REGION Network 174: Reset CV hơi Bồn 4 khi không chạy PID
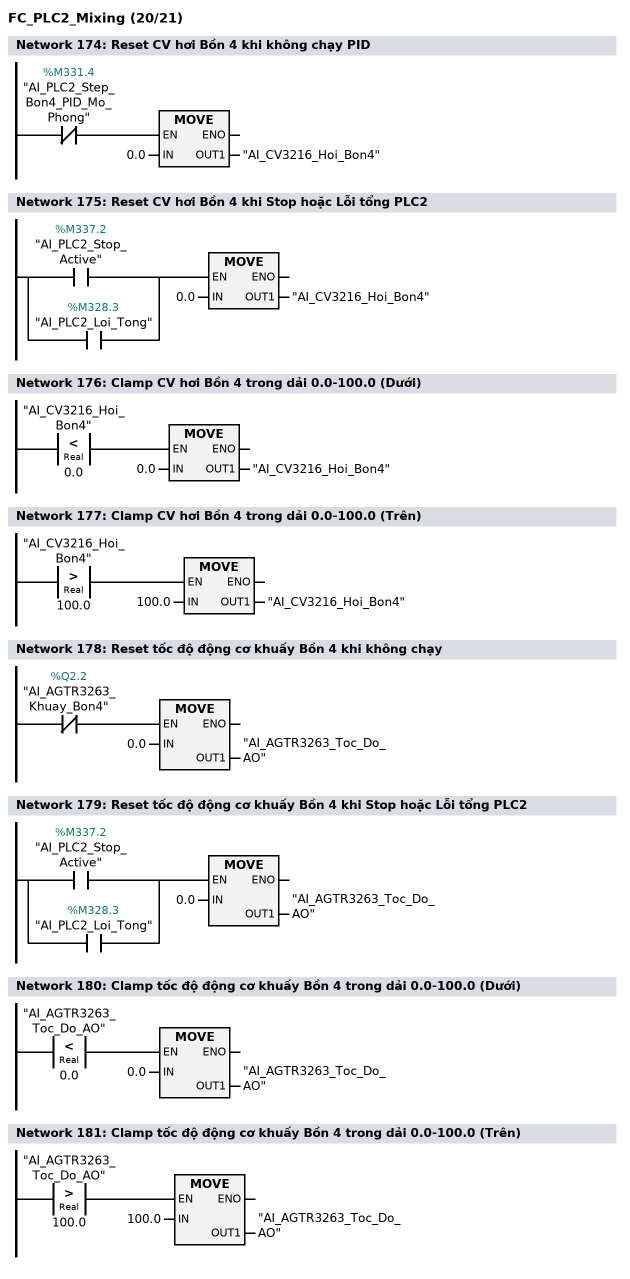
   RUNG wire#powerrail
      I_Contact( "AI_PLC2_Step_Bon4_PID_Mo_Phong" )
      { S7_GenerateENO := "TRUE" } Move(in := 0.0, out1 => "AI_CV3216_Hoi_Bon4")
   END_RUNG
   // the same network as SCL:
   IF NOT "AI_PLC2_Step_Bon4_PID_Mo_Phong" THEN "AI_CV3216_Hoi_Bon4" := 0.0; END_IF;
END_REGION

REGION Network 175: Reset CV hơi Bồn 4 khi Stop hoặc Lỗi tổng PLC2
   RUNG wire#powerrail
      Contact( "AI_PLC2_Stop_Active" )
      wire#w1
      { S7_GenerateENO := "TRUE" } Move(in := 0.0, out1 => "AI_CV3216_Hoi_Bon4")
   END_RUNG
   RUNG wire#powerrail
      Contact( "AI_PLC2_Loi_Tong" )
   END_RUNG wire#w1
   // the same network as SCL:
   IF "AI_PLC2_Stop_Active" OR "AI_PLC2_Loi_Tong" THEN "AI_CV3216_Hoi_Bon4" := 0.0; END_IF;
END_REGION

REGION Network 176: Clamp CV hơi Bồn 4 trong dải 0.0-100.0 (Dưới)
   RUNG wire#powerrail
      { S7_Templates := "SrcType := Real" } LT_Contact(in1 := "AI_CV3216_Hoi_Bon4", in2 := 0.0)
      { S7_GenerateENO := "TRUE" } Move(in := 0.0, out1 => "AI_CV3216_Hoi_Bon4")
   END_RUNG
   // the same network as SCL:
   IF "AI_CV3216_Hoi_Bon4" < 0.0 THEN "AI_CV3216_Hoi_Bon4" := 0.0; END_IF;
END_REGION

REGION Network 177: Clamp CV hơi Bồn 4 trong dải 0.0-100.0 (Trên)
   RUNG wire#powerrail
      { S7_Templates := "SrcType := Real" } GT_Contact(in1 := "AI_CV3216_Hoi_Bon4", in2 := 100.0)
      { S7_GenerateENO := "TRUE" } Move(in := 100.0, out1 => "AI_CV3216_Hoi_Bon4")
   END_RUNG
   // the same network as SCL:
   IF "AI_CV3216_Hoi_Bon4" > 100.0 THEN "AI_CV3216_Hoi_Bon4" := 100.0; END_IF;
END_REGION

REGION Network 178: Reset tốc độ động cơ khuấy Bồn 4 khi không chạy
   RUNG wire#powerrail
      I_Contact( "AI_AGTR3263_Khuay_Bon4" )
      { S7_GenerateENO := "TRUE" } Move(in := 0.0, out1 => "AI_AGTR3263_Toc_Do_AO")
   END_RUNG
   // the same network as SCL:
   IF NOT "AI_AGTR3263_Khuay_Bon4" THEN "AI_AGTR3263_Toc_Do_AO" := 0.0; END_IF;
END_REGION

REGION Network 179: Reset tốc độ động cơ khuấy Bồn 4 khi Stop hoặc Lỗi tổng PLC2
   RUNG wire#powerrail
      Contact( "AI_PLC2_Stop_Active" )
      wire#w1
      { S7_GenerateENO := "TRUE" } Move(in := 0.0, out1 => "AI_AGTR3263_Toc_Do_AO")
   END_RUNG
   RUNG wire#powerrail
      Contact( "AI_PLC2_Loi_Tong" )
   END_RUNG wire#w1
   // the same network as SCL:
   IF "AI_PLC2_Stop_Active" OR "AI_PLC2_Loi_Tong" THEN "AI_AGTR3263_Toc_Do_AO" := 0.0; END_IF;
END_REGION

REGION Network 180: Clamp tốc độ động cơ khuấy Bồn 4 trong dải 0.0-100.0 (Dưới)
   RUNG wire#powerrail
      { S7_Templates := "SrcType := Real" } LT_Contact(in1 := "AI_AGTR3263_Toc_Do_AO", in2 := 0.0)
      { S7_GenerateENO := "TRUE" } Move(in := 0.0, out1 => "AI_AGTR3263_Toc_Do_AO")
   END_RUNG
   // the same network as SCL:
   IF "AI_AGTR3263_Toc_Do_AO" < 0.0 THEN "AI_AGTR3263_Toc_Do_AO" := 0.0; END_IF;
END_REGION

REGION Network 181: Clamp tốc độ động cơ khuấy Bồn 4 trong dải 0.0-100.0 (Trên)
   RUNG wire#powerrail
      { S7_Templates := "SrcType := Real" } GT_Contact(in1 := "AI_AGTR3263_Toc_Do_AO", in2 := 100.0)
      { S7_GenerateENO := "TRUE" } Move(in := 100.0, out1 => "AI_AGTR3263_Toc_Do_AO")
   END_RUNG
   // the same network as SCL:
   IF "AI_AGTR3263_Toc_Do_AO" > 100.0 THEN "AI_AGTR3263_Toc_Do_AO" := 100.0; END_IF;
END_REGION

REGION Network 182: Dừng an toàn PLC2 reset AI_V3240_Nuoc_Bon3
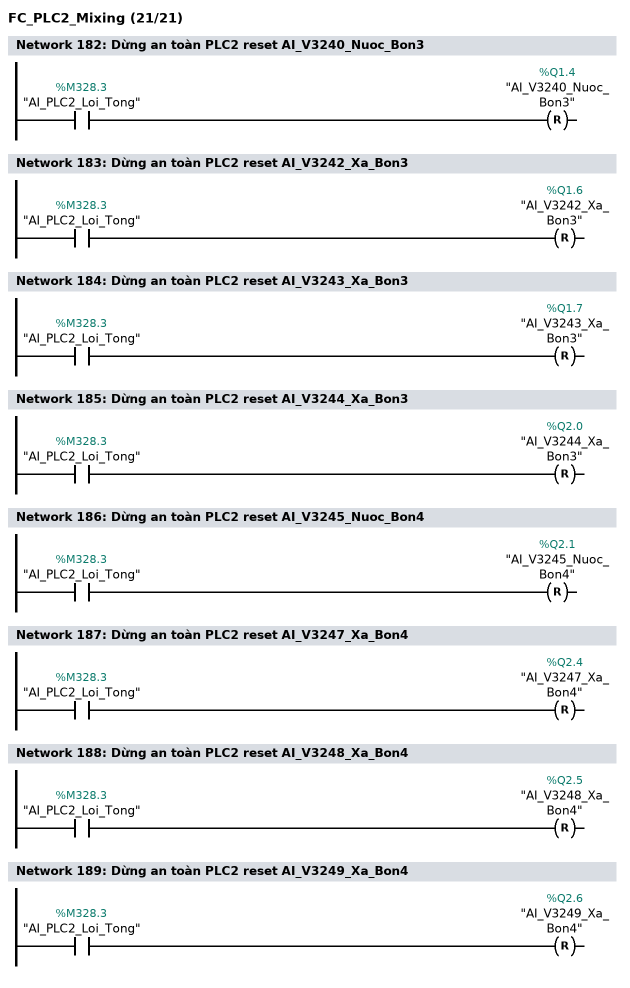
   RUNG wire#powerrail
      Contact( "AI_PLC2_Loi_Tong" )
      R_Coil( "AI_V3240_Nuoc_Bon3" )
   END_RUNG
   // the same network as SCL:
   IF "AI_PLC2_Loi_Tong" THEN "AI_V3240_Nuoc_Bon3" := FALSE; END_IF;
END_REGION

REGION Network 183: Dừng an toàn PLC2 reset AI_V3242_Xa_Bon3
   RUNG wire#powerrail
      Contact( "AI_PLC2_Loi_Tong" )
      R_Coil( "AI_V3242_Xa_Bon3" )
   END_RUNG
   // the same network as SCL:
   IF "AI_PLC2_Loi_Tong" THEN "AI_V3242_Xa_Bon3" := FALSE; END_IF;
END_REGION

REGION Network 184: Dừng an toàn PLC2 reset AI_V3243_Xa_Bon3
   RUNG wire#powerrail
      Contact( "AI_PLC2_Loi_Tong" )
      R_Coil( "AI_V3243_Xa_Bon3" )
   END_RUNG
   // the same network as SCL:
   IF "AI_PLC2_Loi_Tong" THEN "AI_V3243_Xa_Bon3" := FALSE; END_IF;
END_REGION

REGION Network 185: Dừng an toàn PLC2 reset AI_V3244_Xa_Bon3
   RUNG wire#powerrail
      Contact( "AI_PLC2_Loi_Tong" )
      R_Coil( "AI_V3244_Xa_Bon3" )
   END_RUNG
   // the same network as SCL:
   IF "AI_PLC2_Loi_Tong" THEN "AI_V3244_Xa_Bon3" := FALSE; END_IF;
END_REGION

REGION Network 186: Dừng an toàn PLC2 reset AI_V3245_Nuoc_Bon4
   RUNG wire#powerrail
      Contact( "AI_PLC2_Loi_Tong" )
      R_Coil( "AI_V3245_Nuoc_Bon4" )
   END_RUNG
   // the same network as SCL:
   IF "AI_PLC2_Loi_Tong" THEN "AI_V3245_Nuoc_Bon4" := FALSE; END_IF;
END_REGION

REGION Network 187: Dừng an toàn PLC2 reset AI_V3247_Xa_Bon4
   RUNG wire#powerrail
      Contact( "AI_PLC2_Loi_Tong" )
      R_Coil( "AI_V3247_Xa_Bon4" )
   END_RUNG
   // the same network as SCL:
   IF "AI_PLC2_Loi_Tong" THEN "AI_V3247_Xa_Bon4" := FALSE; END_IF;
END_REGION

REGION Network 188: Dừng an toàn PLC2 reset AI_V3248_Xa_Bon4
   RUNG wire#powerrail
      Contact( "AI_PLC2_Loi_Tong" )
      R_Coil( "AI_V3248_Xa_Bon4" )
   END_RUNG
   // the same network as SCL:
   IF "AI_PLC2_Loi_Tong" THEN "AI_V3248_Xa_Bon4" := FALSE; END_IF;
END_REGION

REGION Network 189: Dừng an toàn PLC2 reset AI_V3249_Xa_Bon4
   RUNG wire#powerrail
      Contact( "AI_PLC2_Loi_Tong" )
      R_Coil( "AI_V3249_Xa_Bon4" )
   END_RUNG
   // the same network as SCL:
   IF "AI_PLC2_Loi_Tong" THEN "AI_V3249_Xa_Bon4" := FALSE; END_IF;
END_REGION
END_FUNCTION

FUNCTION "FC_HMI_Mirror_PLC2" : Void   // FC41, LAD
{ S7_Optimized_Access := 'TRUE' }
VERSION : 0.1
// stored: AutoNumber true, IsIECCheckEnabled false, SetENOAutomatically false, UDAEnableTagReadback false
BEGIN

REGION Network 1: Mirror AI_V3240_Nuoc_Bon3
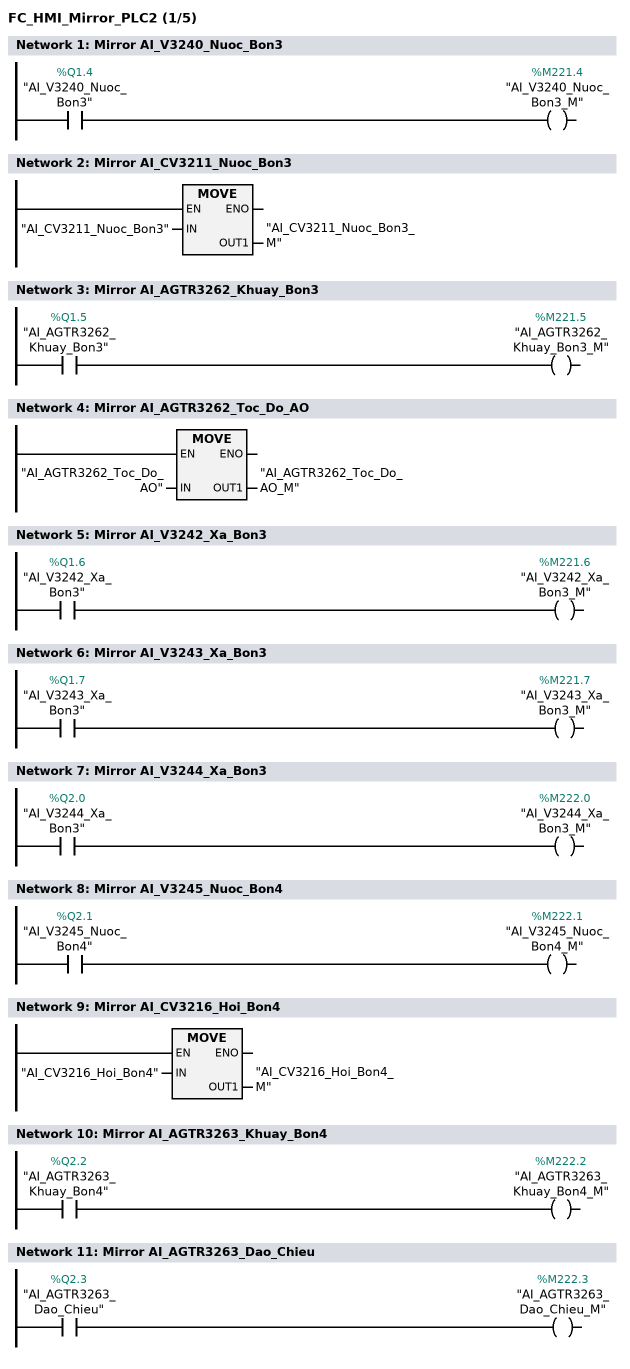
   RUNG wire#powerrail
      Contact( "AI_V3240_Nuoc_Bon3" )
      Coil( "AI_V3240_Nuoc_Bon3_M" )
   END_RUNG
   // the same network as SCL:
   "AI_V3240_Nuoc_Bon3_M" := "AI_V3240_Nuoc_Bon3";
END_REGION

REGION Network 2: Mirror AI_CV3211_Nuoc_Bon3
   RUNG wire#powerrail
      { S7_GenerateENO := "TRUE" } Move(in := "AI_CV3211_Nuoc_Bon3", out1 => "AI_CV3211_Nuoc_Bon3_M")
   END_RUNG
   // the same network as SCL:
   "AI_CV3211_Nuoc_Bon3_M" := "AI_CV3211_Nuoc_Bon3";
END_REGION

REGION Network 3: Mirror AI_AGTR3262_Khuay_Bon3
   RUNG wire#powerrail
      Contact( "AI_AGTR3262_Khuay_Bon3" )
      Coil( "AI_AGTR3262_Khuay_Bon3_M" )
   END_RUNG
   // the same network as SCL:
   "AI_AGTR3262_Khuay_Bon3_M" := "AI_AGTR3262_Khuay_Bon3";
END_REGION

REGION Network 4: Mirror AI_AGTR3262_Toc_Do_AO
   RUNG wire#powerrail
      { S7_GenerateENO := "TRUE" } Move(in := "AI_AGTR3262_Toc_Do_AO", out1 => "AI_AGTR3262_Toc_Do_AO_M")
   END_RUNG
   // the same network as SCL:
   "AI_AGTR3262_Toc_Do_AO_M" := "AI_AGTR3262_Toc_Do_AO";
END_REGION

REGION Network 5: Mirror AI_V3242_Xa_Bon3
   RUNG wire#powerrail
      Contact( "AI_V3242_Xa_Bon3" )
      Coil( "AI_V3242_Xa_Bon3_M" )
   END_RUNG
   // the same network as SCL:
   "AI_V3242_Xa_Bon3_M" := "AI_V3242_Xa_Bon3";
END_REGION

REGION Network 6: Mirror AI_V3243_Xa_Bon3
   RUNG wire#powerrail
      Contact( "AI_V3243_Xa_Bon3" )
      Coil( "AI_V3243_Xa_Bon3_M" )
   END_RUNG
   // the same network as SCL:
   "AI_V3243_Xa_Bon3_M" := "AI_V3243_Xa_Bon3";
END_REGION

REGION Network 7: Mirror AI_V3244_Xa_Bon3
   RUNG wire#powerrail
      Contact( "AI_V3244_Xa_Bon3" )
      Coil( "AI_V3244_Xa_Bon3_M" )
   END_RUNG
   // the same network as SCL:
   "AI_V3244_Xa_Bon3_M" := "AI_V3244_Xa_Bon3";
END_REGION

REGION Network 8: Mirror AI_V3245_Nuoc_Bon4
   RUNG wire#powerrail
      Contact( "AI_V3245_Nuoc_Bon4" )
      Coil( "AI_V3245_Nuoc_Bon4_M" )
   END_RUNG
   // the same network as SCL:
   "AI_V3245_Nuoc_Bon4_M" := "AI_V3245_Nuoc_Bon4";
END_REGION

REGION Network 9: Mirror AI_CV3216_Hoi_Bon4
   RUNG wire#powerrail
      { S7_GenerateENO := "TRUE" } Move(in := "AI_CV3216_Hoi_Bon4", out1 => "AI_CV3216_Hoi_Bon4_M")
   END_RUNG
   // the same network as SCL:
   "AI_CV3216_Hoi_Bon4_M" := "AI_CV3216_Hoi_Bon4";
END_REGION

REGION Network 10: Mirror AI_AGTR3263_Khuay_Bon4
   RUNG wire#powerrail
      Contact( "AI_AGTR3263_Khuay_Bon4" )
      Coil( "AI_AGTR3263_Khuay_Bon4_M" )
   END_RUNG
   // the same network as SCL:
   "AI_AGTR3263_Khuay_Bon4_M" := "AI_AGTR3263_Khuay_Bon4";
END_REGION

REGION Network 11: Mirror AI_AGTR3263_Dao_Chieu
   RUNG wire#powerrail
      Contact( "AI_AGTR3263_Dao_Chieu" )
      Coil( "AI_AGTR3263_Dao_Chieu_M" )
   END_RUNG
   // the same network as SCL:
   "AI_AGTR3263_Dao_Chieu_M" := "AI_AGTR3263_Dao_Chieu";
END_REGION

REGION Network 12: Mirror AI_AGTR3263_Toc_Do_AO
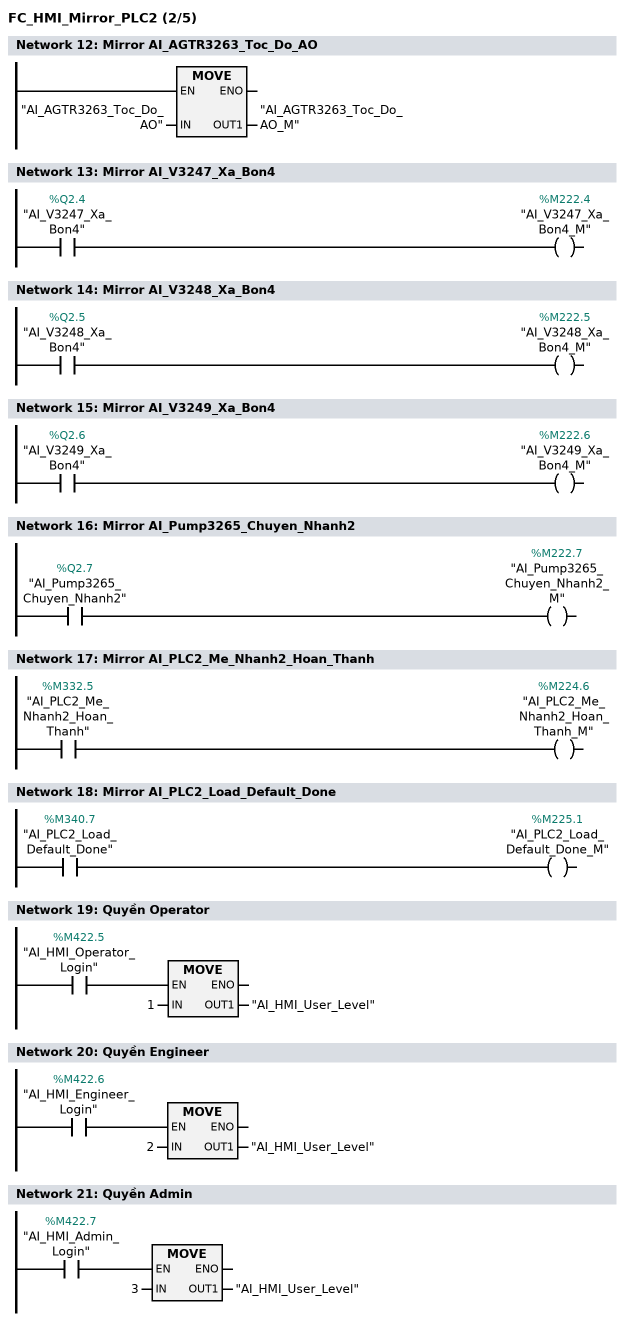
   RUNG wire#powerrail
      { S7_GenerateENO := "TRUE" } Move(in := "AI_AGTR3263_Toc_Do_AO", out1 => "AI_AGTR3263_Toc_Do_AO_M")
   END_RUNG
   // the same network as SCL:
   "AI_AGTR3263_Toc_Do_AO_M" := "AI_AGTR3263_Toc_Do_AO";
END_REGION

REGION Network 13: Mirror AI_V3247_Xa_Bon4
   RUNG wire#powerrail
      Contact( "AI_V3247_Xa_Bon4" )
      Coil( "AI_V3247_Xa_Bon4_M" )
   END_RUNG
   // the same network as SCL:
   "AI_V3247_Xa_Bon4_M" := "AI_V3247_Xa_Bon4";
END_REGION

REGION Network 14: Mirror AI_V3248_Xa_Bon4
   RUNG wire#powerrail
      Contact( "AI_V3248_Xa_Bon4" )
      Coil( "AI_V3248_Xa_Bon4_M" )
   END_RUNG
   // the same network as SCL:
   "AI_V3248_Xa_Bon4_M" := "AI_V3248_Xa_Bon4";
END_REGION

REGION Network 15: Mirror AI_V3249_Xa_Bon4
   RUNG wire#powerrail
      Contact( "AI_V3249_Xa_Bon4" )
      Coil( "AI_V3249_Xa_Bon4_M" )
   END_RUNG
   // the same network as SCL:
   "AI_V3249_Xa_Bon4_M" := "AI_V3249_Xa_Bon4";
END_REGION

REGION Network 16: Mirror AI_Pump3265_Chuyen_Nhanh2
   RUNG wire#powerrail
      Contact( "AI_Pump3265_Chuyen_Nhanh2" )
      Coil( "AI_Pump3265_Chuyen_Nhanh2_M" )
   END_RUNG
   // the same network as SCL:
   "AI_Pump3265_Chuyen_Nhanh2_M" := "AI_Pump3265_Chuyen_Nhanh2";
END_REGION

REGION Network 17: Mirror AI_PLC2_Me_Nhanh2_Hoan_Thanh
   RUNG wire#powerrail
      Contact( "AI_PLC2_Me_Nhanh2_Hoan_Thanh" )
      Coil( "AI_PLC2_Me_Nhanh2_Hoan_Thanh_M" )
   END_RUNG
   // the same network as SCL:
   "AI_PLC2_Me_Nhanh2_Hoan_Thanh_M" := "AI_PLC2_Me_Nhanh2_Hoan_Thanh";
END_REGION

REGION Network 18: Mirror AI_PLC2_Load_Default_Done
   RUNG wire#powerrail
      Contact( "AI_PLC2_Load_Default_Done" )
      Coil( "AI_PLC2_Load_Default_Done_M" )
   END_RUNG
   // the same network as SCL:
   "AI_PLC2_Load_Default_Done_M" := "AI_PLC2_Load_Default_Done";
END_REGION

REGION Network 19: Quyền Operator
   RUNG wire#powerrail
      Contact( "AI_HMI_Operator_Login" )
      { S7_GenerateENO := "TRUE" } Move(in := 1, out1 => "AI_HMI_User_Level")
   END_RUNG
   // the same network as SCL:
   IF "AI_HMI_Operator_Login" THEN "AI_HMI_User_Level" := 1; END_IF;
END_REGION

REGION Network 20: Quyền Engineer
   RUNG wire#powerrail
      Contact( "AI_HMI_Engineer_Login" )
      { S7_GenerateENO := "TRUE" } Move(in := 2, out1 => "AI_HMI_User_Level")
   END_RUNG
   // the same network as SCL:
   IF "AI_HMI_Engineer_Login" THEN "AI_HMI_User_Level" := 2; END_IF;
END_REGION

REGION Network 21: Quyền Admin
   RUNG wire#powerrail
      Contact( "AI_HMI_Admin_Login" )
      { S7_GenerateENO := "TRUE" } Move(in := 3, out1 => "AI_HMI_User_Level")
   END_RUNG
   // the same network as SCL:
   IF "AI_HMI_Admin_Login" THEN "AI_HMI_User_Level" := 3; END_IF;
END_REGION

REGION Network 22: Cho phép sửa thông số Engineer
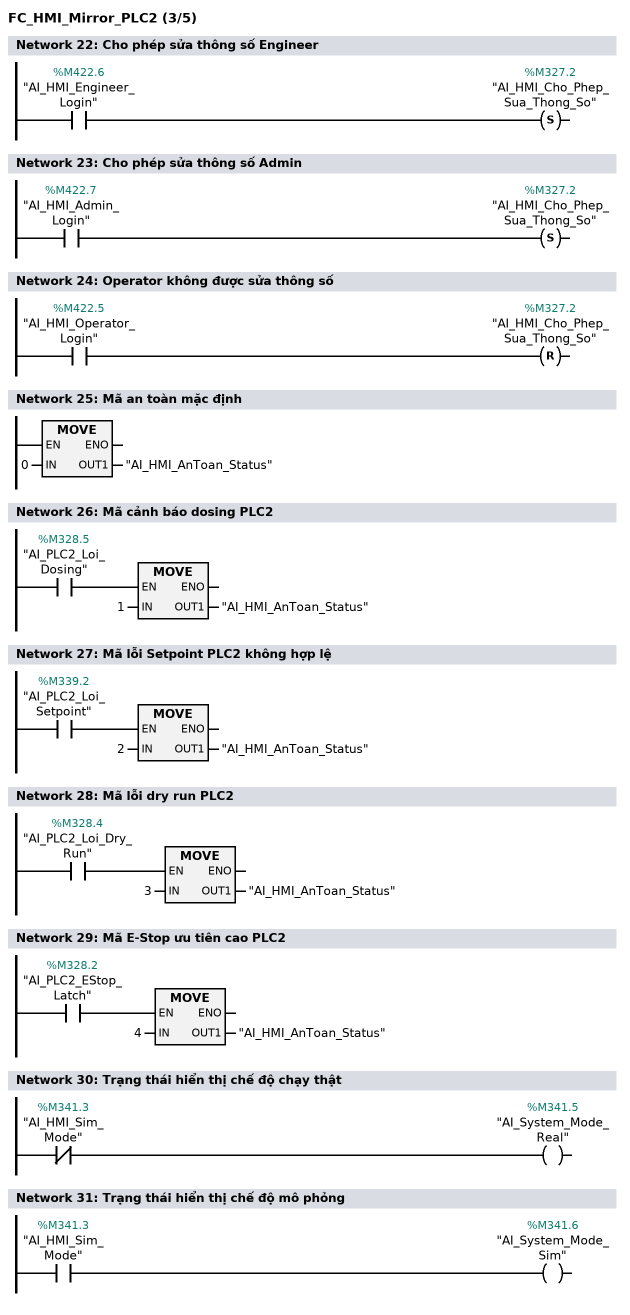
   RUNG wire#powerrail
      Contact( "AI_HMI_Engineer_Login" )
      S_Coil( "AI_HMI_Cho_Phep_Sua_Thong_So" )
   END_RUNG
   // the same network as SCL:
   IF "AI_HMI_Engineer_Login" THEN "AI_HMI_Cho_Phep_Sua_Thong_So" := TRUE; END_IF;
END_REGION

REGION Network 23: Cho phép sửa thông số Admin
   RUNG wire#powerrail
      Contact( "AI_HMI_Admin_Login" )
      S_Coil( "AI_HMI_Cho_Phep_Sua_Thong_So" )
   END_RUNG
   // the same network as SCL:
   IF "AI_HMI_Admin_Login" THEN "AI_HMI_Cho_Phep_Sua_Thong_So" := TRUE; END_IF;
END_REGION

REGION Network 24: Operator không được sửa thông số
   RUNG wire#powerrail
      Contact( "AI_HMI_Operator_Login" )
      R_Coil( "AI_HMI_Cho_Phep_Sua_Thong_So" )
   END_RUNG
   // the same network as SCL:
   IF "AI_HMI_Operator_Login" THEN "AI_HMI_Cho_Phep_Sua_Thong_So" := FALSE; END_IF;
END_REGION

REGION Network 25: Mã an toàn mặc định
   RUNG wire#powerrail
      { S7_GenerateENO := "TRUE" } Move(in := 0, out1 => "AI_HMI_AnToan_Status")
   END_RUNG
   // the same network as SCL:
   "AI_HMI_AnToan_Status" := 0;
END_REGION

REGION Network 26: Mã cảnh báo dosing PLC2
   RUNG wire#powerrail
      Contact( "AI_PLC2_Loi_Dosing" )
      { S7_GenerateENO := "TRUE" } Move(in := 1, out1 => "AI_HMI_AnToan_Status")
   END_RUNG
   // the same network as SCL:
   IF "AI_PLC2_Loi_Dosing" THEN "AI_HMI_AnToan_Status" := 1; END_IF;
END_REGION

REGION Network 27: Mã lỗi Setpoint PLC2 không hợp lệ
   RUNG wire#powerrail
      Contact( "AI_PLC2_Loi_Setpoint" )
      { S7_GenerateENO := "TRUE" } Move(in := 2, out1 => "AI_HMI_AnToan_Status")
   END_RUNG
   // the same network as SCL:
   IF "AI_PLC2_Loi_Setpoint" THEN "AI_HMI_AnToan_Status" := 2; END_IF;
END_REGION

REGION Network 28: Mã lỗi dry run PLC2
   RUNG wire#powerrail
      Contact( "AI_PLC2_Loi_Dry_Run" )
      { S7_GenerateENO := "TRUE" } Move(in := 3, out1 => "AI_HMI_AnToan_Status")
   END_RUNG
   // the same network as SCL:
   IF "AI_PLC2_Loi_Dry_Run" THEN "AI_HMI_AnToan_Status" := 3; END_IF;
END_REGION

REGION Network 29: Mã E-Stop ưu tiên cao PLC2
   RUNG wire#powerrail
      Contact( "AI_PLC2_EStop_Latch" )
      { S7_GenerateENO := "TRUE" } Move(in := 4, out1 => "AI_HMI_AnToan_Status")
   END_RUNG
   // the same network as SCL:
   IF "AI_PLC2_EStop_Latch" THEN "AI_HMI_AnToan_Status" := 4; END_IF;
END_REGION

REGION Network 30: Trạng thái hiển thị chế độ chạy thật
   RUNG wire#powerrail
      I_Contact( "AI_HMI_Sim_Mode" )
      Coil( "AI_System_Mode_Real" )
   END_RUNG
   // the same network as SCL:
   "AI_System_Mode_Real" := NOT "AI_HMI_Sim_Mode";
END_REGION

REGION Network 31: Trạng thái hiển thị chế độ mô phỏng
   RUNG wire#powerrail
      Contact( "AI_HMI_Sim_Mode" )
      Coil( "AI_System_Mode_Sim" )
   END_RUNG
   // the same network as SCL:
   "AI_System_Mode_Sim" := "AI_HMI_Sim_Mode";
END_REGION

REGION Network 32: Cảnh báo chế độ mô phỏng HMI active
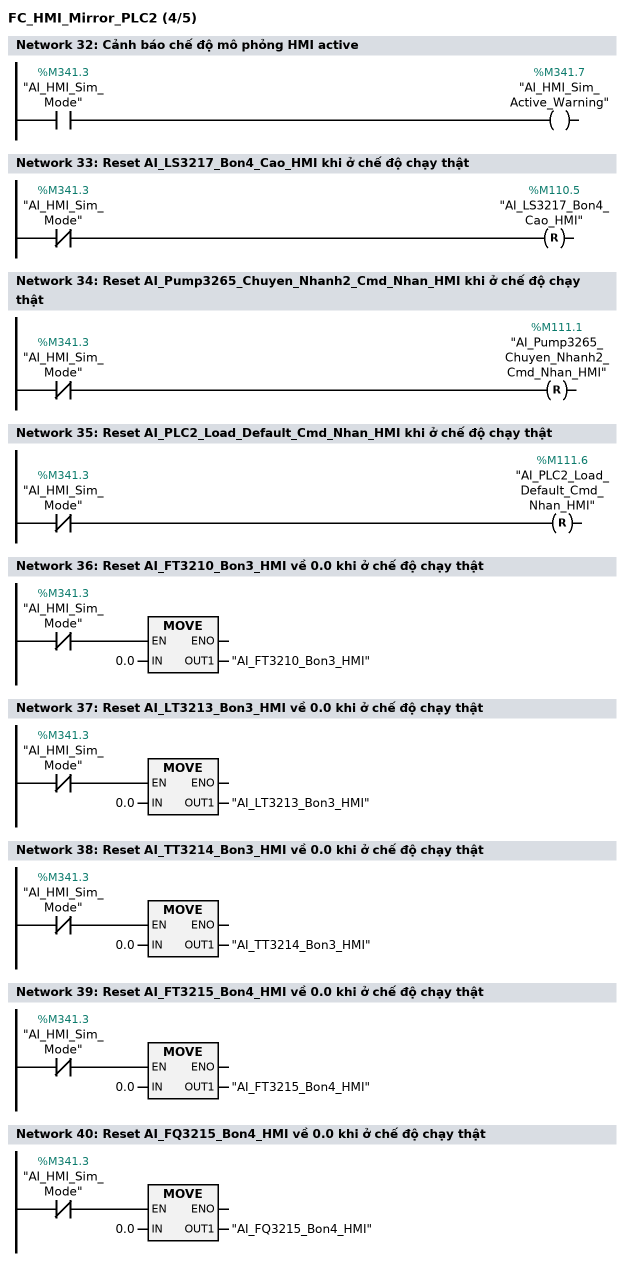
   RUNG wire#powerrail
      Contact( "AI_HMI_Sim_Mode" )
      Coil( "AI_HMI_Sim_Active_Warning" )
   END_RUNG
   // the same network as SCL:
   "AI_HMI_Sim_Active_Warning" := "AI_HMI_Sim_Mode";
END_REGION

REGION Network 33: Reset AI_LS3217_Bon4_Cao_HMI khi ở chế độ chạy thật
   RUNG wire#powerrail
      I_Contact( "AI_HMI_Sim_Mode" )
      R_Coil( "AI_LS3217_Bon4_Cao_HMI" )
   END_RUNG
   // the same network as SCL:
   IF NOT "AI_HMI_Sim_Mode" THEN "AI_LS3217_Bon4_Cao_HMI" := FALSE; END_IF;
END_REGION

REGION Network 34: Reset AI_Pump3265_Chuyen_Nhanh2_Cmd_Nhan_HMI khi ở chế độ chạy thật
   RUNG wire#powerrail
      I_Contact( "AI_HMI_Sim_Mode" )
      R_Coil( "AI_Pump3265_Chuyen_Nhanh2_Cmd_Nhan_HMI" )
   END_RUNG
   // the same network as SCL:
   IF NOT "AI_HMI_Sim_Mode" THEN "AI_Pump3265_Chuyen_Nhanh2_Cmd_Nhan_HMI" := FALSE; END_IF;
END_REGION

REGION Network 35: Reset AI_PLC2_Load_Default_Cmd_Nhan_HMI khi ở chế độ chạy thật
   RUNG wire#powerrail
      I_Contact( "AI_HMI_Sim_Mode" )
      R_Coil( "AI_PLC2_Load_Default_Cmd_Nhan_HMI" )
   END_RUNG
   // the same network as SCL:
   IF NOT "AI_HMI_Sim_Mode" THEN "AI_PLC2_Load_Default_Cmd_Nhan_HMI" := FALSE; END_IF;
END_REGION

REGION Network 36: Reset AI_FT3210_Bon3_HMI về 0.0 khi ở chế độ chạy thật
   RUNG wire#powerrail
      I_Contact( "AI_HMI_Sim_Mode" )
      { S7_GenerateENO := "TRUE" } Move(in := 0.0, out1 => "AI_FT3210_Bon3_HMI")
   END_RUNG
   // the same network as SCL:
   IF NOT "AI_HMI_Sim_Mode" THEN "AI_FT3210_Bon3_HMI" := 0.0; END_IF;
END_REGION

REGION Network 37: Reset AI_LT3213_Bon3_HMI về 0.0 khi ở chế độ chạy thật
   RUNG wire#powerrail
      I_Contact( "AI_HMI_Sim_Mode" )
      { S7_GenerateENO := "TRUE" } Move(in := 0.0, out1 => "AI_LT3213_Bon3_HMI")
   END_RUNG
   // the same network as SCL:
   IF NOT "AI_HMI_Sim_Mode" THEN "AI_LT3213_Bon3_HMI" := 0.0; END_IF;
END_REGION

REGION Network 38: Reset AI_TT3214_Bon3_HMI về 0.0 khi ở chế độ chạy thật
   RUNG wire#powerrail
      I_Contact( "AI_HMI_Sim_Mode" )
      { S7_GenerateENO := "TRUE" } Move(in := 0.0, out1 => "AI_TT3214_Bon3_HMI")
   END_RUNG
   // the same network as SCL:
   IF NOT "AI_HMI_Sim_Mode" THEN "AI_TT3214_Bon3_HMI" := 0.0; END_IF;
END_REGION

REGION Network 39: Reset AI_FT3215_Bon4_HMI về 0.0 khi ở chế độ chạy thật
   RUNG wire#powerrail
      I_Contact( "AI_HMI_Sim_Mode" )
      { S7_GenerateENO := "TRUE" } Move(in := 0.0, out1 => "AI_FT3215_Bon4_HMI")
   END_RUNG
   // the same network as SCL:
   IF NOT "AI_HMI_Sim_Mode" THEN "AI_FT3215_Bon4_HMI" := 0.0; END_IF;
END_REGION

REGION Network 40: Reset AI_FQ3215_Bon4_HMI về 0.0 khi ở chế độ chạy thật
   RUNG wire#powerrail
      I_Contact( "AI_HMI_Sim_Mode" )
      { S7_GenerateENO := "TRUE" } Move(in := 0.0, out1 => "AI_FQ3215_Bon4_HMI")
   END_RUNG
   // the same network as SCL:
   IF NOT "AI_HMI_Sim_Mode" THEN "AI_FQ3215_Bon4_HMI" := 0.0; END_IF;
END_REGION

REGION Network 41: Reset AI_LT3218_Bon4_HMI về 0.0 khi ở chế độ chạy thật
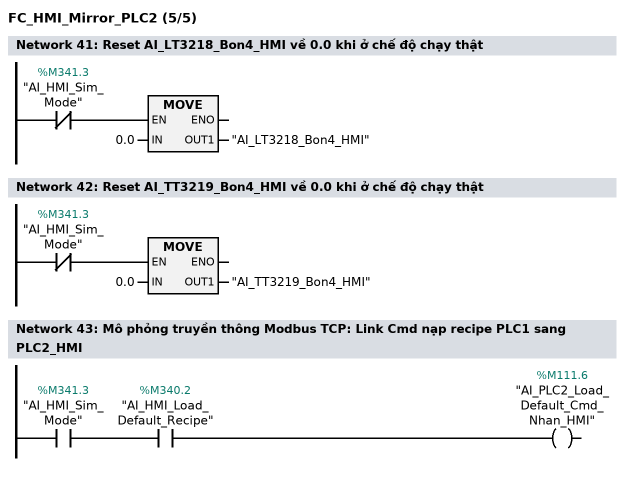
   RUNG wire#powerrail
      I_Contact( "AI_HMI_Sim_Mode" )
      { S7_GenerateENO := "TRUE" } Move(in := 0.0, out1 => "AI_LT3218_Bon4_HMI")
   END_RUNG
   // the same network as SCL:
   IF NOT "AI_HMI_Sim_Mode" THEN "AI_LT3218_Bon4_HMI" := 0.0; END_IF;
END_REGION

REGION Network 42: Reset AI_TT3219_Bon4_HMI về 0.0 khi ở chế độ chạy thật
   RUNG wire#powerrail
      I_Contact( "AI_HMI_Sim_Mode" )
      { S7_GenerateENO := "TRUE" } Move(in := 0.0, out1 => "AI_TT3219_Bon4_HMI")
   END_RUNG
   // the same network as SCL:
   IF NOT "AI_HMI_Sim_Mode" THEN "AI_TT3219_Bon4_HMI" := 0.0; END_IF;
END_REGION

REGION Network 43: Mô phỏng truyền thông Modbus TCP: Link Cmd nạp recipe PLC1 sang PLC2_HMI
   RUNG wire#powerrail
      Contact( "AI_HMI_Sim_Mode" )
      Contact( "AI_HMI_Load_Default_Recipe" )
      Coil( "AI_PLC2_Load_Default_Cmd_Nhan_HMI" )
   END_RUNG
   // the same network as SCL:
   "AI_PLC2_Load_Default_Cmd_Nhan_HMI" := "AI_HMI_Sim_Mode" AND "AI_HMI_Load_Default_Recipe";
END_REGION
END_FUNCTION

ORGANIZATION_BLOCK "OB31_PID_PLC2_Bon4"   // OB31, LAD, CyclicInterrupt
{ S7_Optimized_Access := 'TRUE' }
VERSION : 0.1
// stored: AutoNumber true, IsIECCheckEnabled false, SetENOAutomatically false
   VAR_INPUT
      Initial_Call : Bool;   // Initial call of this OB
      Event_Count : Int;   // Events discarded
   END_VAR
BEGIN

REGION Network 1: Initialize PID Bon 4 Kp parameter
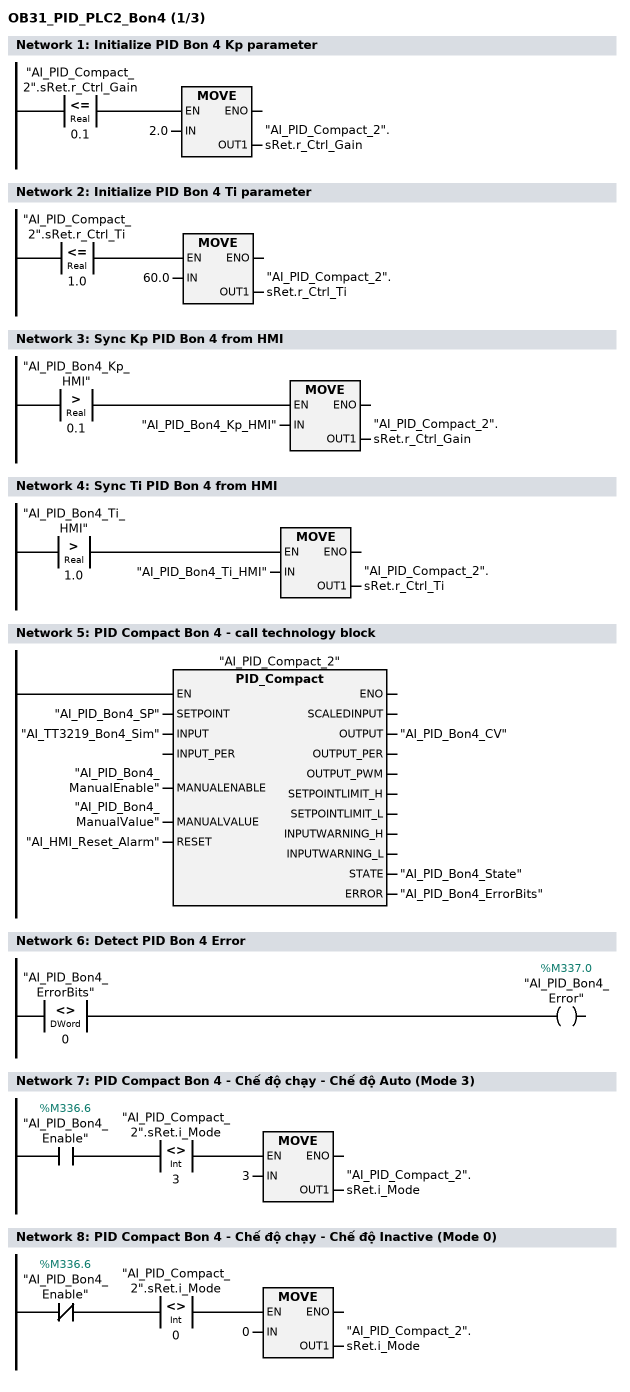
   RUNG wire#powerrail
      { S7_Templates := "SrcType := Real" } LE_Contact(in1 := "AI_PID_Compact_2".sRet.r_Ctrl_Gain, in2 := 0.1)
      { S7_GenerateENO := "TRUE" } Move(in := 2.0, out1 => "AI_PID_Compact_2".sRet.r_Ctrl_Gain)
   END_RUNG
   // the same network as SCL:
   IF "AI_PID_Compact_2".sRet.r_Ctrl_Gain <= 0.1 THEN "AI_PID_Compact_2".sRet.r_Ctrl_Gain := 2.0; END_IF;
END_REGION

REGION Network 2: Initialize PID Bon 4 Ti parameter
   RUNG wire#powerrail
      { S7_Templates := "SrcType := Real" } LE_Contact(in1 := "AI_PID_Compact_2".sRet.r_Ctrl_Ti, in2 := 1.0)
      { S7_GenerateENO := "TRUE" } Move(in := 60.0, out1 => "AI_PID_Compact_2".sRet.r_Ctrl_Ti)
   END_RUNG
   // the same network as SCL:
   IF "AI_PID_Compact_2".sRet.r_Ctrl_Ti <= 1.0 THEN "AI_PID_Compact_2".sRet.r_Ctrl_Ti := 60.0; END_IF;
END_REGION

REGION Network 3: Sync Kp PID Bon 4 from HMI
   RUNG wire#powerrail
      { S7_Templates := "SrcType := Real" } GT_Contact(in1 := "AI_PID_Bon4_Kp_HMI", in2 := 0.1)
      { S7_GenerateENO := "TRUE" } Move(in := "AI_PID_Bon4_Kp_HMI", out1 => "AI_PID_Compact_2".sRet.r_Ctrl_Gain)
   END_RUNG
   // the same network as SCL:
   IF "AI_PID_Bon4_Kp_HMI" > 0.1 THEN "AI_PID_Compact_2".sRet.r_Ctrl_Gain := "AI_PID_Bon4_Kp_HMI"; END_IF;
END_REGION

REGION Network 4: Sync Ti PID Bon 4 from HMI
   RUNG wire#powerrail
      { S7_Templates := "SrcType := Real" } GT_Contact(in1 := "AI_PID_Bon4_Ti_HMI", in2 := 1.0)
      { S7_GenerateENO := "TRUE" } Move(in := "AI_PID_Bon4_Ti_HMI", out1 => "AI_PID_Compact_2".sRet.r_Ctrl_Ti)
   END_RUNG
   // the same network as SCL:
   IF "AI_PID_Bon4_Ti_HMI" > 1.0 THEN "AI_PID_Compact_2".sRet.r_Ctrl_Ti := "AI_PID_Bon4_Ti_HMI"; END_IF;
END_REGION

REGION Network 5: PID Compact Bon 4 - call technology block
   RUNG wire#powerrail
      "AI_PID_Compact_2".PID_Compact(Setpoint := "AI_PID_Bon4_SP", Input := "AI_TT3219_Bon4_Sim", Input_PER :=, ManualEnable := "AI_PID_Bon4_ManualEnable", ManualValue := "AI_PID_Bon4_ManualValue", Reset := "AI_HMI_Reset_Alarm", ScaledInput =>, Output => "AI_PID_Bon4_CV", Output_PER =>, Output_PWM =>, SetpointLimit_H =>, SetpointLimit_L =>, InputWarning_H =>, InputWarning_L =>, State => "AI_PID_Bon4_State", Error => "AI_PID_Bon4_ErrorBits")
   END_RUNG
   // the same network as SCL:
   "AI_PID_Compact_2"(Setpoint := "AI_PID_Bon4_SP",   // PID_Compact
                      Input := "AI_TT3219_Bon4_Sim",
                      ManualEnable := "AI_PID_Bon4_ManualEnable",
                      ManualValue := "AI_PID_Bon4_ManualValue",
                      Reset := "AI_HMI_Reset_Alarm",
                      Output => "AI_PID_Bon4_CV",
                      State => "AI_PID_Bon4_State",
                      Error => "AI_PID_Bon4_ErrorBits");
END_REGION

REGION Network 6: Detect PID Bon 4 Error
   RUNG wire#powerrail
      { S7_Templates := "SrcType := DWord" } NE_Contact(in1 := "AI_PID_Bon4_ErrorBits", in2 := 0)
      Coil( "AI_PID_Bon4_Error" )
   END_RUNG
   // the same network as SCL:
   "AI_PID_Bon4_Error" := "AI_PID_Bon4_ErrorBits" <> 0;
END_REGION

REGION Network 7: PID Compact Bon 4 - Chế độ chạy - Chế độ Auto (Mode 3)
   RUNG wire#powerrail
      Contact( "AI_PID_Bon4_Enable" )
      { S7_Templates := "SrcType := Int" } NE_Contact(in1 := "AI_PID_Compact_2".sRet.i_Mode, in2 := 3)
      { S7_GenerateENO := "TRUE" } Move(in := 3, out1 => "AI_PID_Compact_2".sRet.i_Mode)
   END_RUNG
   // the same network as SCL:
   IF "AI_PID_Bon4_Enable" AND ("AI_PID_Compact_2".sRet.i_Mode <> 3) THEN
       "AI_PID_Compact_2".sRet.i_Mode := 3;
   END_IF;
END_REGION

REGION Network 8: PID Compact Bon 4 - Chế độ chạy - Chế độ Inactive (Mode 0)
   RUNG wire#powerrail
      I_Contact( "AI_PID_Bon4_Enable" )
      { S7_Templates := "SrcType := Int" } NE_Contact(in1 := "AI_PID_Compact_2".sRet.i_Mode, in2 := 0)
      { S7_GenerateENO := "TRUE" } Move(in := 0, out1 => "AI_PID_Compact_2".sRet.i_Mode)
   END_RUNG
   // the same network as SCL:
   IF NOT "AI_PID_Bon4_Enable" AND ("AI_PID_Compact_2".sRet.i_Mode <> 0) THEN
       "AI_PID_Compact_2".sRet.i_Mode := 0;
   END_IF;
END_REGION

REGION Network 9: Move PID Bon 4 CV to simulated heat valve
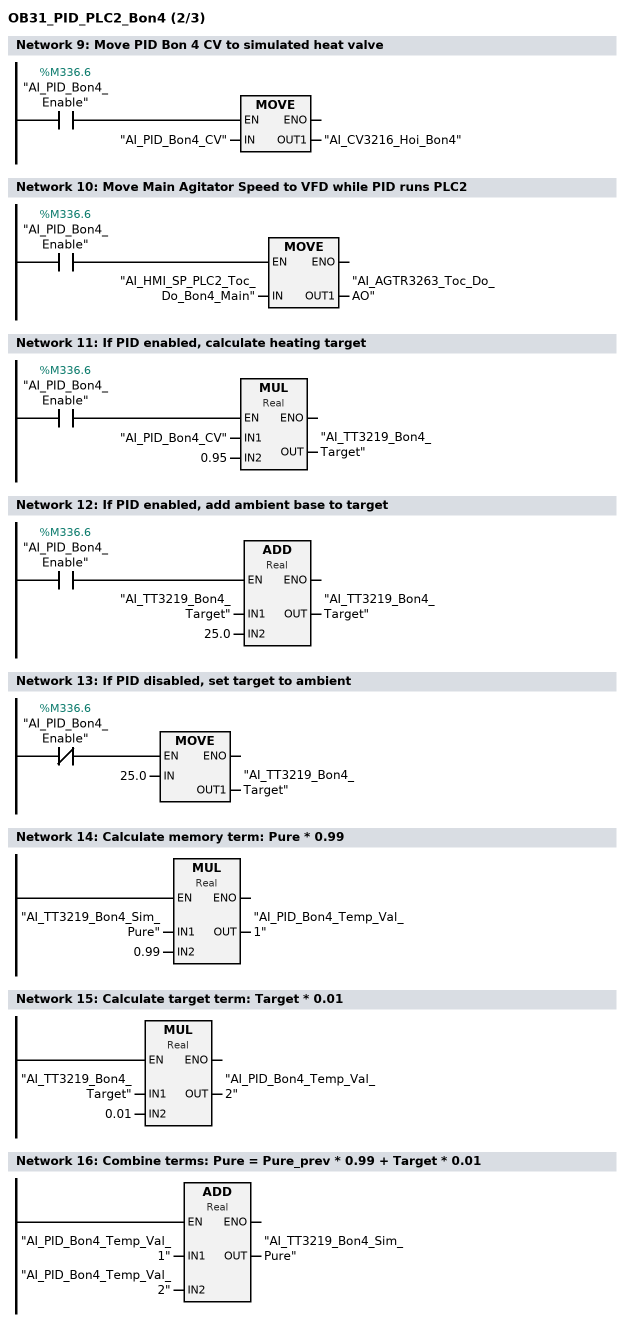
   RUNG wire#powerrail
      Contact( "AI_PID_Bon4_Enable" )
      { S7_GenerateENO := "TRUE" } Move(in := "AI_PID_Bon4_CV", out1 => "AI_CV3216_Hoi_Bon4")
   END_RUNG
   // the same network as SCL:
   IF "AI_PID_Bon4_Enable" THEN "AI_CV3216_Hoi_Bon4" := "AI_PID_Bon4_CV"; END_IF;
END_REGION

REGION Network 10: Move Main Agitator Speed to VFD while PID runs PLC2
   RUNG wire#powerrail
      Contact( "AI_PID_Bon4_Enable" )
      { S7_GenerateENO := "TRUE" } Move(in := "AI_HMI_SP_PLC2_Toc_Do_Bon4_Main", out1 => "AI_AGTR3263_Toc_Do_AO")
   END_RUNG
   // the same network as SCL:
   IF "AI_PID_Bon4_Enable" THEN "AI_AGTR3263_Toc_Do_AO" := "AI_HMI_SP_PLC2_Toc_Do_Bon4_Main"; END_IF;
END_REGION

REGION Network 11: If PID enabled, calculate heating target
   RUNG wire#powerrail
      Contact( "AI_PID_Bon4_Enable" )
      { S7_Templates := "SrcType := Real"; S7_GenerateENO := "TRUE" } Mul(in1 := "AI_PID_Bon4_CV", in2 := 0.95, out => "AI_TT3219_Bon4_Target")
   END_RUNG
   // the same network as SCL:
   IF "AI_PID_Bon4_Enable" THEN "AI_TT3219_Bon4_Target" := "AI_PID_Bon4_CV" * 0.95; END_IF;
END_REGION

REGION Network 12: If PID enabled, add ambient base to target
   RUNG wire#powerrail
      Contact( "AI_PID_Bon4_Enable" )
      { S7_Templates := "SrcType := Real"; S7_GenerateENO := "TRUE" } Add(in1 := "AI_TT3219_Bon4_Target", in2 := 25.0, out => "AI_TT3219_Bon4_Target")
   END_RUNG
   // the same network as SCL:
   IF "AI_PID_Bon4_Enable" THEN "AI_TT3219_Bon4_Target" := "AI_TT3219_Bon4_Target" + 25.0; END_IF;
END_REGION

REGION Network 13: If PID disabled, set target to ambient
   RUNG wire#powerrail
      I_Contact( "AI_PID_Bon4_Enable" )
      { S7_GenerateENO := "TRUE" } Move(in := 25.0, out1 => "AI_TT3219_Bon4_Target")
   END_RUNG
   // the same network as SCL:
   IF NOT "AI_PID_Bon4_Enable" THEN "AI_TT3219_Bon4_Target" := 25.0; END_IF;
END_REGION

REGION Network 14: Calculate memory term: Pure * 0.99
   RUNG wire#powerrail
      { S7_Templates := "SrcType := Real"; S7_GenerateENO := "TRUE" } Mul(in1 := "AI_TT3219_Bon4_Sim_Pure", in2 := 0.99, out => "AI_PID_Bon4_Temp_Val_1")
   END_RUNG
   // the same network as SCL:
   "AI_PID_Bon4_Temp_Val_1" := "AI_TT3219_Bon4_Sim_Pure" * 0.99;
END_REGION

REGION Network 15: Calculate target term: Target * 0.01
   RUNG wire#powerrail
      { S7_Templates := "SrcType := Real"; S7_GenerateENO := "TRUE" } Mul(in1 := "AI_TT3219_Bon4_Target", in2 := 0.01, out => "AI_PID_Bon4_Temp_Val_2")
   END_RUNG
   // the same network as SCL:
   "AI_PID_Bon4_Temp_Val_2" := "AI_TT3219_Bon4_Target" * 0.01;
END_REGION

REGION Network 16: Combine terms: Pure = Pure_prev * 0.99 + Target * 0.01
   RUNG wire#powerrail
      { S7_Templates := "SrcType := Real"; S7_GenerateENO := "TRUE" } Add(in1 := "AI_PID_Bon4_Temp_Val_1", in2 := "AI_PID_Bon4_Temp_Val_2", out => "AI_TT3219_Bon4_Sim_Pure")
   END_RUNG
   // the same network as SCL:
   "AI_TT3219_Bon4_Sim_Pure" := "AI_PID_Bon4_Temp_Val_1" + "AI_PID_Bon4_Temp_Val_2";
END_REGION

REGION Network 17: Increment simulation counter
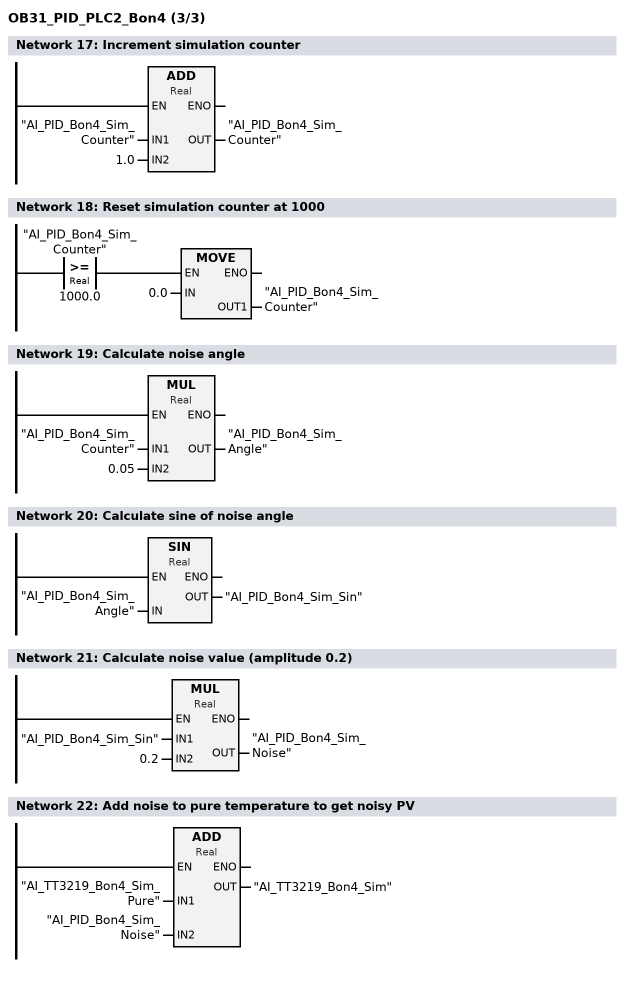
   RUNG wire#powerrail
      { S7_Templates := "SrcType := Real"; S7_GenerateENO := "TRUE" } Add(in1 := "AI_PID_Bon4_Sim_Counter", in2 := 1.0, out => "AI_PID_Bon4_Sim_Counter")
   END_RUNG
   // the same network as SCL:
   "AI_PID_Bon4_Sim_Counter" := "AI_PID_Bon4_Sim_Counter" + 1.0;
END_REGION

REGION Network 18: Reset simulation counter at 1000
   RUNG wire#powerrail
      { S7_Templates := "SrcType := Real" } GE_Contact(in1 := "AI_PID_Bon4_Sim_Counter", in2 := 1000.0)
      { S7_GenerateENO := "TRUE" } Move(in := 0.0, out1 => "AI_PID_Bon4_Sim_Counter")
   END_RUNG
   // the same network as SCL:
   IF "AI_PID_Bon4_Sim_Counter" >= 1000.0 THEN "AI_PID_Bon4_Sim_Counter" := 0.0; END_IF;
END_REGION

REGION Network 19: Calculate noise angle
   RUNG wire#powerrail
      { S7_Templates := "SrcType := Real"; S7_GenerateENO := "TRUE" } Mul(in1 := "AI_PID_Bon4_Sim_Counter", in2 := 0.05, out => "AI_PID_Bon4_Sim_Angle")
   END_RUNG
   // the same network as SCL:
   "AI_PID_Bon4_Sim_Angle" := "AI_PID_Bon4_Sim_Counter" * 0.05;
END_REGION

REGION Network 20: Calculate sine of noise angle
   "AI_PID_Bon4_Sim_Sin" := SIN("AI_PID_Bon4_Sim_Angle");
END_REGION

REGION Network 21: Calculate noise value (amplitude 0.2)
   RUNG wire#powerrail
      { S7_Templates := "SrcType := Real"; S7_GenerateENO := "TRUE" } Mul(in1 := "AI_PID_Bon4_Sim_Sin", in2 := 0.2, out => "AI_PID_Bon4_Sim_Noise")
   END_RUNG
   // the same network as SCL:
   "AI_PID_Bon4_Sim_Noise" := "AI_PID_Bon4_Sim_Sin" * 0.2;
END_REGION

REGION Network 22: Add noise to pure temperature to get noisy PV
   RUNG wire#powerrail
      { S7_Templates := "SrcType := Real"; S7_GenerateENO := "TRUE" } Add(in1 := "AI_TT3219_Bon4_Sim_Pure", in2 := "AI_PID_Bon4_Sim_Noise", out => "AI_TT3219_Bon4_Sim")
   END_RUNG
   // the same network as SCL:
   "AI_TT3219_Bon4_Sim" := "AI_TT3219_Bon4_Sim_Pure" + "AI_PID_Bon4_Sim_Noise";
END_REGION
END_ORGANIZATION_BLOCK

DATA_BLOCK "MB_SERVER_DB"   // DB53
// stored: AutoNumber true, DBAccessibleFromOPCUA true, InstanceOfName MB_SERVER, OfSystemLibElement MB_SERVER, OfSystemLibVersion 3.1
"MB_SERVER"
   // VAR_INPUT
   //    DISCONNECT : Bool;
   //    CONNECT_ID : UInt;
   //    IP_PORT : UInt;
   // END_VAR
   // VAR_OUTPUT
   //    NDR : Bool;
   //    DR : Bool;
   //    ERROR : Bool;
   //    STATUS : Word;
   // END_VAR
   // VAR_IN_OUT
   //    MB_HOLD_REG : Variant;
   // END_VAR
   // VAR
   //    TCON_SFB { S7_SetPoint := 'True'} : TCON;
   //    TDISCON_SFB { S7_SetPoint := 'True'} : TDISCON;
   //    TSEND_SFB { S7_SetPoint := 'True'} : TSEND;
   //    TRCV_SFB { S7_SetPoint := 'True'} : TRCV;
   //    TCON_Param { S7_SetPoint := 'True'} : TCON_Param;
   //    MB_State : UInt;
   //    Request_Count : UInt;
   //    Server_Message_Count : UInt;
   //    Xmt_Rcv_Count : UInt;
   //    Exception_Count : UInt;
   //    Success_Count : UInt;
   //    SL_Status_Hold : UInt;
   //    HR_Start_Offset : UInt;
   //    Init_OK : Bool;
   //    SL_Error_State : Bool;
   //    Connected : Bool;
   //    XMT_Set_NDR : Bool;
   //    XMT_Set_DR : Bool;
   // END_VAR
BEGIN
   TCON_Param.CONNECTION_TYPE := 11;
   TCON_Param.LOCAL_DEVICE_ID := 64;
END_DATA_BLOCK
